TYPE "SubProcessParameterP020_ShW"
VERSION : 0.1
   STRUCT
      Reserved : Bool;
   END_STRUCT;

END_TYPE

